(* Logix 5000 project; controller Laser_Cutter vendor 1 type 14 code 149 rev 28.11; software revision 28.00; part 2 of 4 *)
(* tags used below, declared in another part *)
   aBlowOffOnSol : BOOL;
   aBlowoffTimer : TIMER;
   aBoltDriverDownSol : BOOL;
   aBoltDriverUpSol : BOOL;
   aCameraTrigger : BOOL;
   aDoorSafetySwitchUnlockSol : BOOL;
   aExhaustStart : BOOL;
   alarmActive : BOOL;
   automaticSeqStep : DINT;
   autoMode : BOOL;
   autoModeReady : BOOL;
   aWalkingBeamDownSol : BOOL;
   blowoffSeqStep : DINT;
   boltDriverDownDB : TIMER;
   boltDriverSeqStep : DINT;
   boltDriverToStartPOS : BOOL;
   boltDriverToStartPOSdb : TIMER;
   boltDriverUpDB : TIMER;
   Counter : DINT;
   Counter2 : DINT;
   Counter3 : DINT;
   CYCLE_IN_PROG : BOOL;
   cycleTimer : TIMER;
   exeBlowoffSR : BOOL;
   Exec_Bolt_Driver_SR : BOOL;
   Exec_Drive_Bolt : BOOL;
   Exec_Laser_SR : BOOL;
   execLoadPalletSR : BOOL;
   Execute_BlowoffSR : BOOL;
   Execute_MoveToZoneSR : BOOL;
   Execute_VisionInspectionSR : BOOL;
   executeInitializationSequence : BOOL;
   INIT_START_PB : BOOL;
   initDelayTimer : TIMER;
   inspectionSeqStep : DINT;
   LaserSeqStep : INT;
   loadPalletSeqStep : INT;
   MoveToZoneSeqStep : INT;
   p2pCycleTime : TIMER;
   p2pCycleTimeBuffer : DINT;
   readyToMovePallet : BOOL;
   readyToStartCycle : BOOL;
   rejectPartSR : DINT[1];
   runsCompleted : DINT;
   runTime : TIMER;
   startCycleTimer : BOOL;
   startP2PTimer : BOOL;
   startRunTimer : BOOL;
   stationNumber : CONTROL;
   systemInInitializedPosition : BOOL;
   cameraBadPart : ALIAS FOR Local:1:I.Data.8;
   cameraGoodPart : ALIAS FOR Local:1:I.Data.7;
   collarAtStation3 : ALIAS FOR MURR_IMPACT_IO_1:I.Data[1].0;
   collarAtStation4 : ALIAS FOR MURR_IMPACT_IO_1:I.Data[1].1;
   cycleStartPB : ALIAS FOR Local:1:I.Data.3;
   doorOpenedSafetyRelayStatus : ALIAS FOR Local:1:I.Data.1;
   eStopSafetyRelayStatus : ALIAS FOR Local:1:I.Data.0;
   stopPB : ALIAS FOR Local:1:I.Data.4;
(* MainProgram, continued *)

ROUTINE Auto_Seq   (* ladder *)
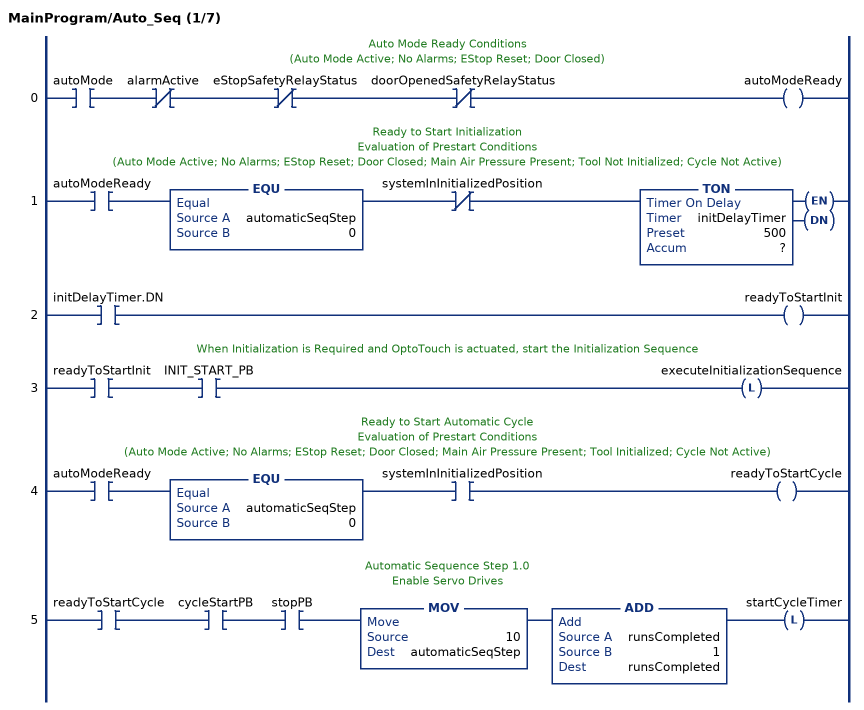
   // Auto Mode Ready Conditions
   // (Auto Mode Active; No Alarms; EStop Reset; Door Closed)
   0: XIC(autoMode)XIO(alarmActive)XIO(eStopSafetyRelayStatus)XIO(doorOpenedSafetyRelayStatus)OTE(autoModeReady);
   // Ready to Start Initialization
   // Evaluation of Prestart Conditions
   // (Auto Mode Active; No Alarms; EStop Reset; Door Closed; Main Air Pressure Present; Tool Not Initialized; Cycle Not Active)
   1: XIC(autoModeReady)EQU(automaticSeqStep,0)XIO(systemInInitializedPosition)TON(initDelayTimer,?,?);
   2: XIC(initDelayTimer.DN)OTE(readyToStartInit);
   // When Initialization is Required and OptoTouch is actuated, start the Initialization Sequence
   3: XIC(readyToStartInit)XIC(INIT_START_PB)OTL(executeInitializationSequence);
   // Ready to Start Automatic Cycle
   // Evaluation of Prestart Conditions
   // (Auto Mode Active; No Alarms; EStop Reset; Door Closed; Main Air Pressure Present; Tool Initialized; Cycle Not Active)
   4: XIC(autoModeReady)EQU(automaticSeqStep,0)XIC(systemInInitializedPosition)OTE(readyToStartCycle);
   // Automatic Sequence Step 1.0
   // Enable Servo Drives
   5: XIC(readyToStartCycle)XIC(cycleStartPB)XIC(stopPB)MOV(10,automaticSeqStep)ADD(runsCompleted,1,runsCompleted)OTL(startCycleTimer);
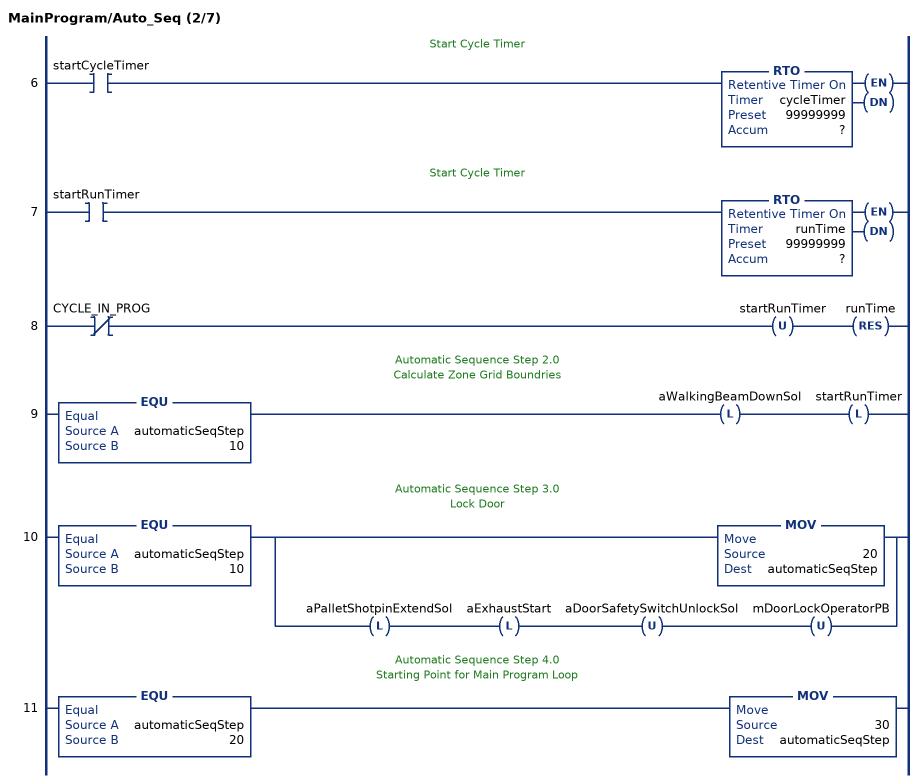
   // Start Cycle Timer
   6: XIC(startCycleTimer)RTO(cycleTimer,?,?);
   // Start Cycle Timer
   7: XIC(startRunTimer)RTO(runTime,?,?);
   8: XIO(CYCLE_IN_PROG)OTU(startRunTimer)RES(runTime);
   // Automatic Sequence Step 2.0
   // Calculate Zone Grid Boundries
   9: EQU(automaticSeqStep,10)OTL(aWalkingBeamDownSol)OTL(startRunTimer);
   // Automatic Sequence Step 3.0
   // Lock Door
   10: EQU(automaticSeqStep,10)[MOV(20,automaticSeqStep) ,OTL(aPalletShotpinExtendSol) OTL(aExhaustStart) OTU(aDoorSafetySwitchUnlockSol) OTU(mDoorLockOperatorPB) ];
   // Automatic Sequence Step 4.0
   // Starting Point for Main Program Loop
   11: EQU(automaticSeqStep,20)MOV(30,automaticSeqStep);
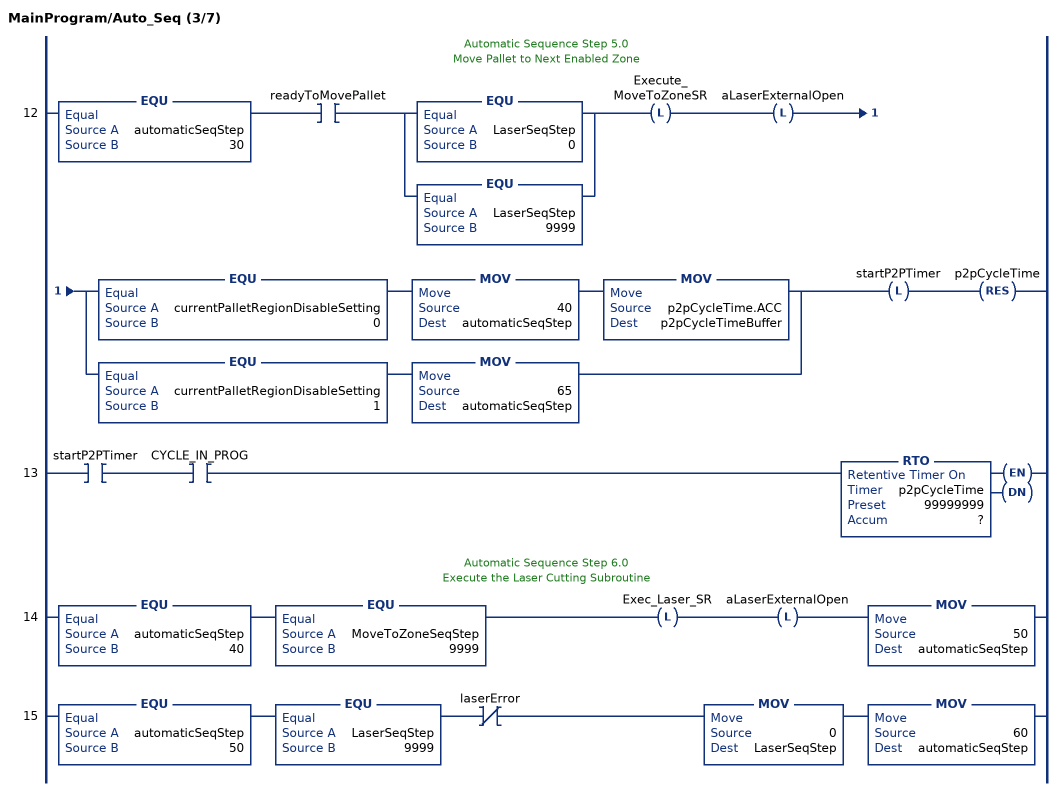
   // Automatic Sequence Step 5.0
   // Move Pallet to Next Enabled Zone
   12: EQU(automaticSeqStep,30)XIC(readyToMovePallet)[EQU(LaserSeqStep,0) ,EQU(LaserSeqStep,9999) ]OTL(Execute_MoveToZoneSR)OTL(aLaserExternalOpen)[EQU(currentPalletRegionDisableSetting,0) MOV(40,automaticSeqStep) MOV(p2pCycleTime.ACC,p2pCycleTimeBuffer) ,EQU(currentPalletRegionDisableSetting,1) MOV(65,automaticSeqStep) ]OTL(startP2PTimer)RES(p2pCycleTime);
   13: XIC(startP2PTimer)XIC(CYCLE_IN_PROG)RTO(p2pCycleTime,?,?);
   // Automatic Sequence Step 6.0
   // Execute the Laser Cutting Subroutine
   14: EQU(automaticSeqStep,40)EQU(MoveToZoneSeqStep,9999)OTL(Exec_Laser_SR)OTL(aLaserExternalOpen)MOV(50,automaticSeqStep);
   15: EQU(automaticSeqStep,50)EQU(LaserSeqStep,9999)XIO(laserError)MOV(0,LaserSeqStep)MOV(60,automaticSeqStep);
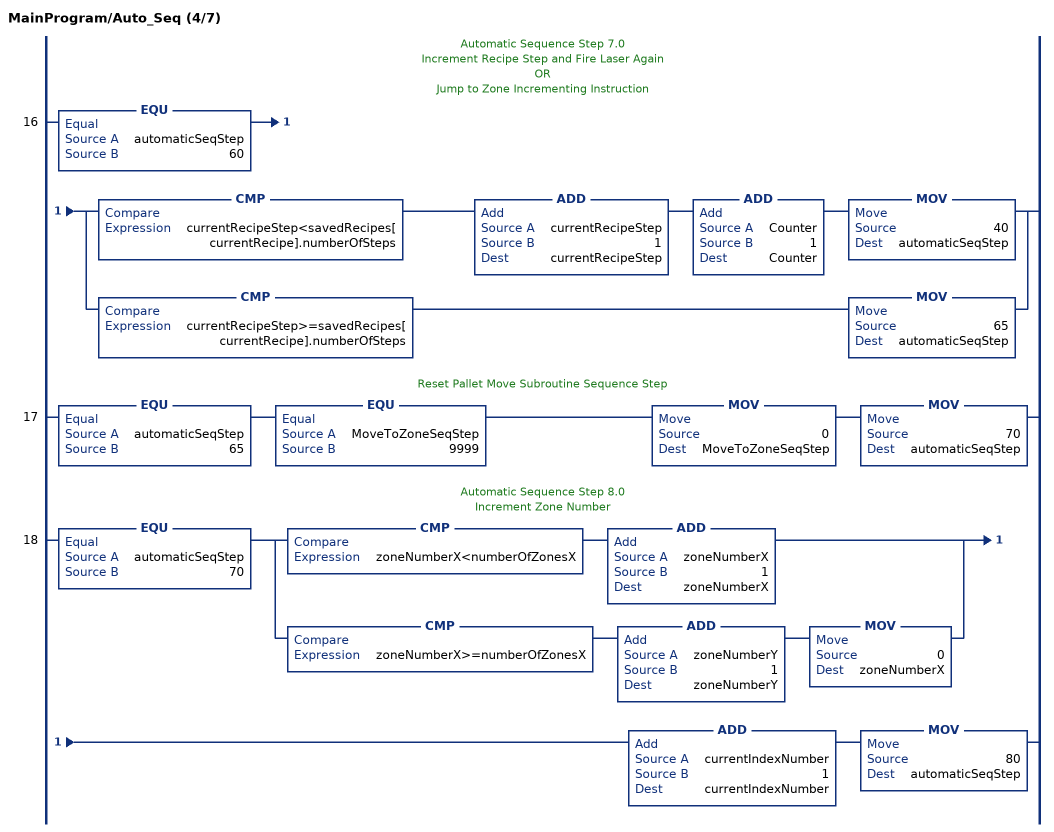
   // Automatic Sequence Step 7.0
   // Increment Recipe Step and Fire Laser Again
   // OR
   // Jump to Zone Incrementing Instruction
   16: EQU(automaticSeqStep,60)[CMP(currentRecipeStep<savedRecipes[currentRecipe].numberOfSteps) ADD(currentRecipeStep,1,currentRecipeStep) ADD(Counter,1,Counter) MOV(40,automaticSeqStep) ,CMP(currentRecipeStep>=savedRecipes[currentRecipe].numberOfSteps) MOV(65,automaticSeqStep) ];
   // Reset Pallet Move Subroutine Sequence Step
   17: EQU(automaticSeqStep,65)EQU(MoveToZoneSeqStep,9999)MOV(0,MoveToZoneSeqStep)MOV(70,automaticSeqStep);
   // Automatic Sequence Step 8.0
   // Increment Zone Number
   18: EQU(automaticSeqStep,70)[CMP(zoneNumberX<numberOfZonesX) ADD(zoneNumberX,1,zoneNumberX) ,CMP(zoneNumberX>=numberOfZonesX) ADD(zoneNumberY,1,zoneNumberY) MOV(0,zoneNumberX) ]ADD(currentIndexNumber,1,currentIndexNumber)MOV(80,automaticSeqStep);
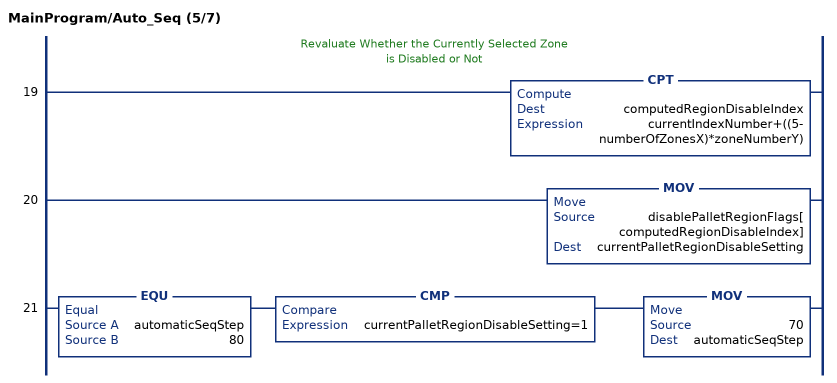
   // Revaluate Whether the Currently Selected Zone
   // is Disabled or Not
   19: CPT(computedRegionDisableIndex,currentIndexNumber+((5-numberOfZonesX)*zoneNumberY));
   20: MOV(disablePalletRegionFlags[computedRegionDisableIndex],currentPalletRegionDisableSetting);
   21: EQU(automaticSeqStep,80)CMP(currentPalletRegionDisableSetting=1)MOV(70,automaticSeqStep);
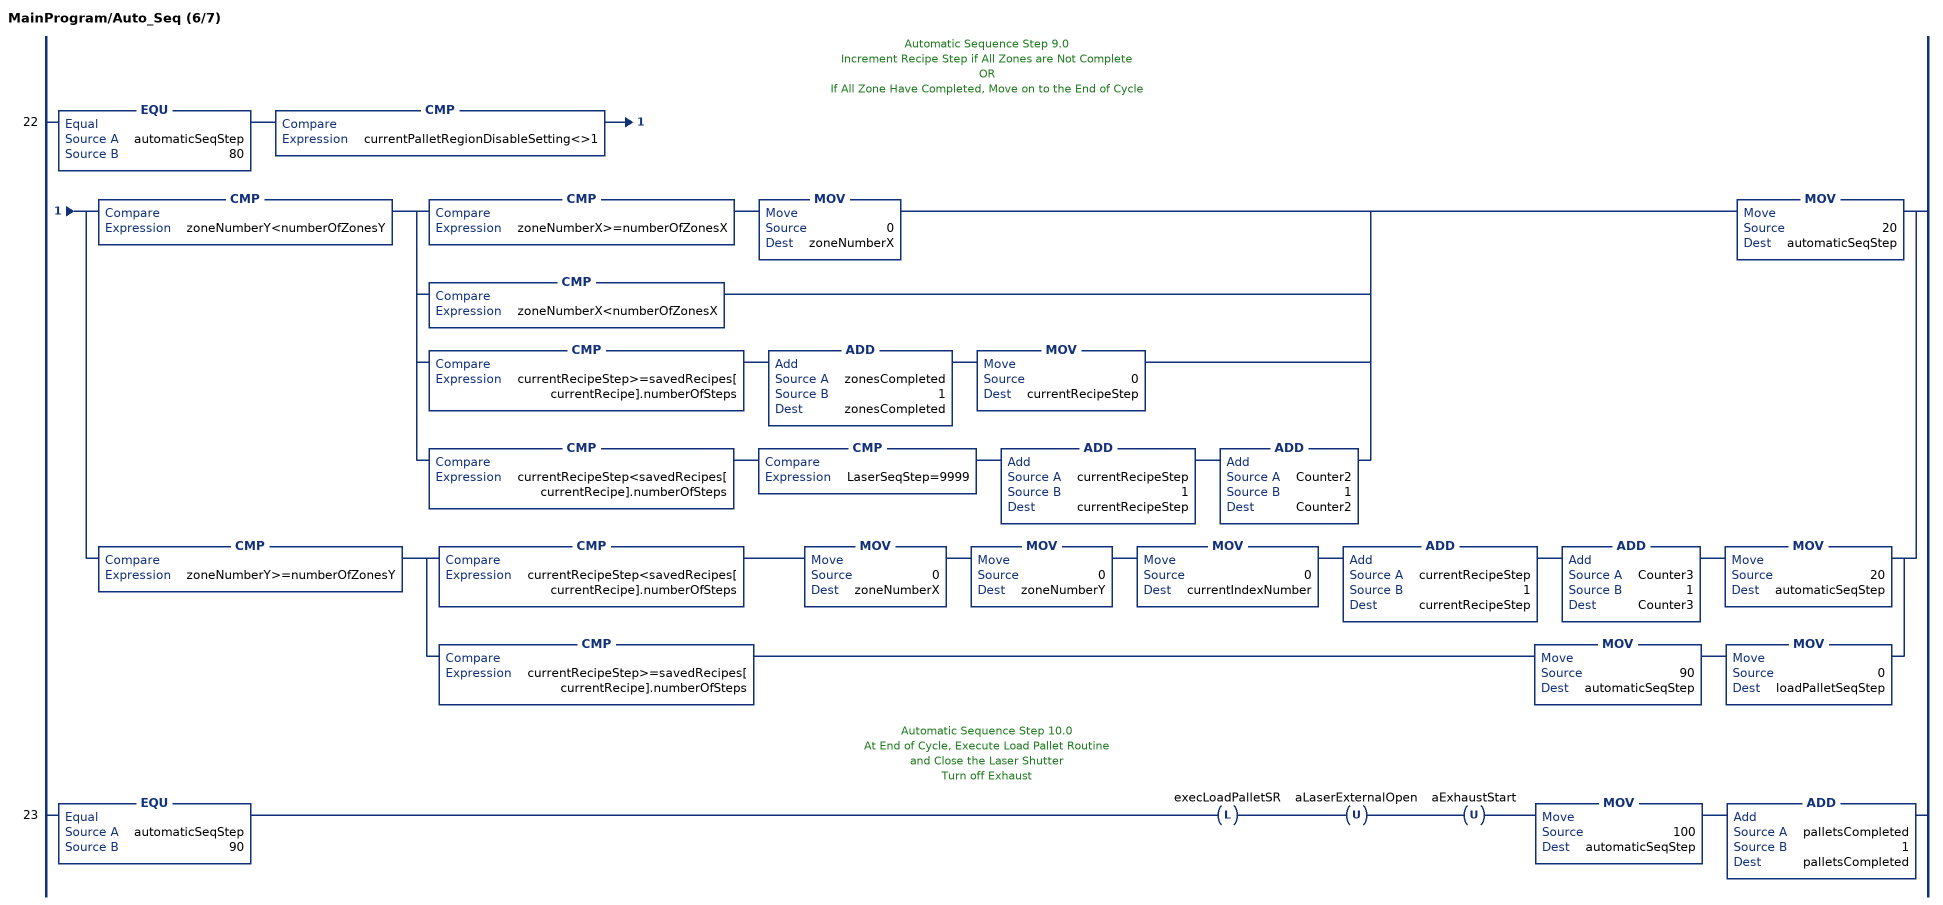
   // Automatic Sequence Step 9.0
   // Increment Recipe Step if All Zones are Not Complete
   // OR
   // If All Zone Have Completed, Move on to the End of Cycle
   22: EQU(automaticSeqStep,80)CMP(currentPalletRegionDisableSetting<>1)[CMP(zoneNumberY<numberOfZonesY) [CMP(zoneNumberX>=numberOfZonesX) MOV(0,zoneNumberX) ,CMP(zoneNumberX<numberOfZonesX) ,[CMP(currentRecipeStep>=savedRecipes[currentRecipe].numberOfSteps) ADD(zonesCompleted,1,zonesCompleted) MOV(0,currentRecipeStep) ,CMP(currentRecipeStep<savedRecipes[currentRecipe].numberOfSteps) CMP(LaserSeqStep=9999) ADD(currentRecipeStep,1,currentRecipeStep) ADD(Counter2,1,Counter2) ] ] MOV(20,automaticSeqStep) ,CMP(zoneNumberY>=numberOfZonesY) [CMP(currentRecipeStep<savedRecipes[currentRecipe].numberOfSteps) MOV(0,zoneNumberX) MOV(0,zoneNumberY) MOV(0,currentIndexNumber) ADD(currentRecipeStep,1,currentRecipeStep) ADD(Counter3,1,Counter3) MOV(20,automaticSeqStep) ,CMP(currentRecipeStep>=savedRecipes[currentRecipe].numberOfSteps) MOV(90,automaticSeqStep) MOV(0,loadPalletSeqStep) ] ];
   // Automatic Sequence Step 10.0
   // At End of Cycle, Execute Load Pallet Routine
   // and Close the Laser Shutter
   // Turn off Exhaust
   23: EQU(automaticSeqStep,90)OTL(execLoadPalletSR)OTU(aLaserExternalOpen)OTU(aExhaustStart)MOV(100,automaticSeqStep)ADD(palletsCompleted,1,palletsCompleted);
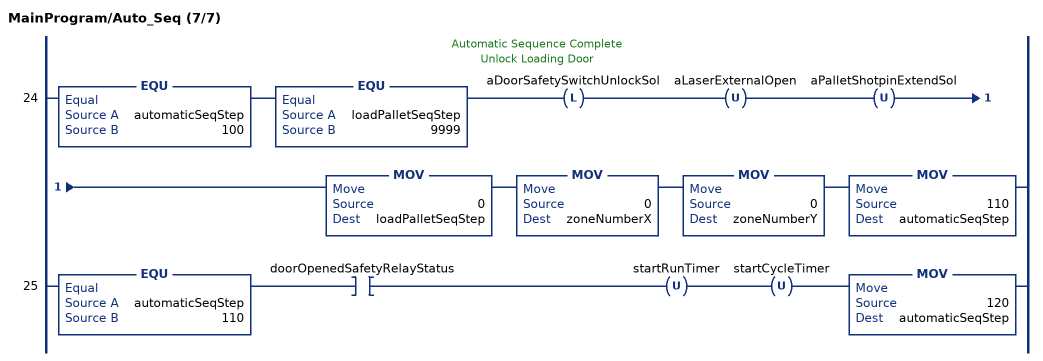
   // Automatic Sequence Complete
   // Unlock Loading Door
   24: EQU(automaticSeqStep,100)EQU(loadPalletSeqStep,9999)OTL(aDoorSafetySwitchUnlockSol)OTU(aLaserExternalOpen)OTU(aPalletShotpinExtendSol)MOV(0,loadPalletSeqStep)MOV(0,zoneNumberX)MOV(0,zoneNumberY)MOV(110,automaticSeqStep);
   25: EQU(automaticSeqStep,110)XIC(doorOpenedSafetyRelayStatus)OTU(startRunTimer)OTU(startCycleTimer)MOV(120,automaticSeqStep);
END_ROUTINE

ROUTINE CycleStations   (* ladder *)
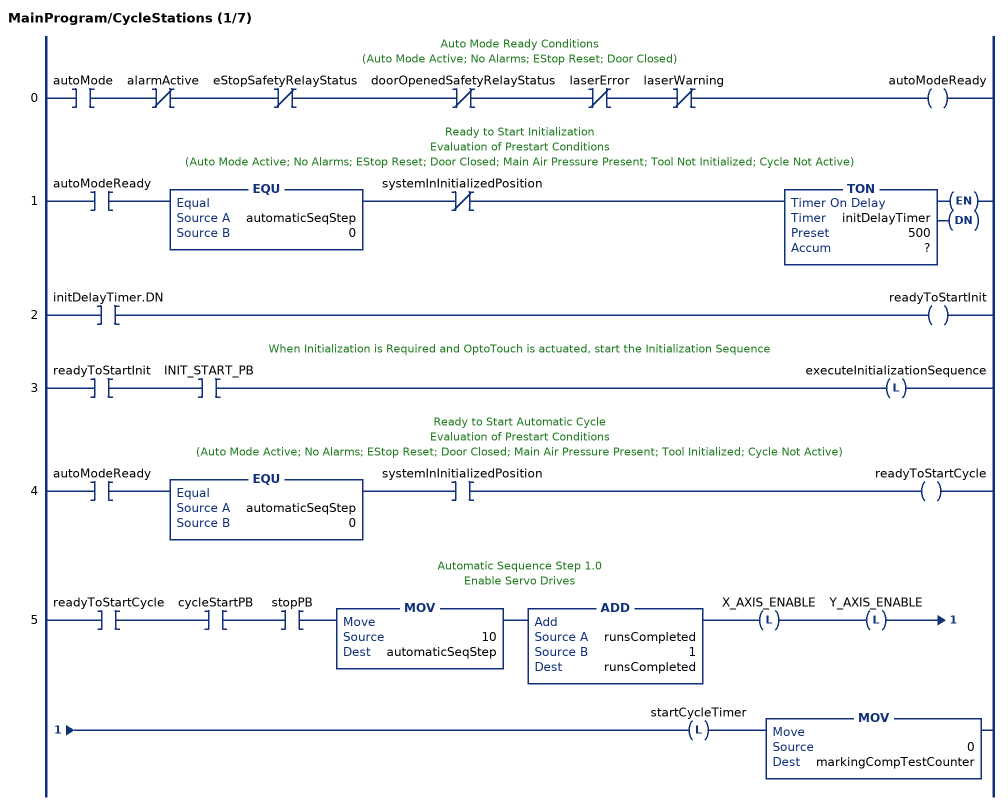
   // Auto Mode Ready Conditions
   // (Auto Mode Active; No Alarms; EStop Reset; Door Closed)
   0: XIC(autoMode)XIO(alarmActive)XIO(eStopSafetyRelayStatus)XIO(doorOpenedSafetyRelayStatus)XIO(laserError)XIO(laserWarning)OTE(autoModeReady);
   // Ready to Start Initialization
   // Evaluation of Prestart Conditions
   // (Auto Mode Active; No Alarms; EStop Reset; Door Closed; Main Air Pressure Present; Tool Not Initialized; Cycle Not Active)
   1: XIC(autoModeReady)EQU(automaticSeqStep,0)XIO(systemInInitializedPosition)TON(initDelayTimer,?,?);
   2: XIC(initDelayTimer.DN)OTE(readyToStartInit);
   // When Initialization is Required and OptoTouch is actuated, start the Initialization Sequence
   3: XIC(readyToStartInit)XIC(INIT_START_PB)OTL(executeInitializationSequence);
   // Ready to Start Automatic Cycle
   // Evaluation of Prestart Conditions
   // (Auto Mode Active; No Alarms; EStop Reset; Door Closed; Main Air Pressure Present; Tool Initialized; Cycle Not Active)
   4: XIC(autoModeReady)EQU(automaticSeqStep,0)XIC(systemInInitializedPosition)OTE(readyToStartCycle);
   // Automatic Sequence Step 1.0
   // Enable Servo Drives
   5: XIC(readyToStartCycle)XIC(cycleStartPB)XIC(stopPB)MOV(10,automaticSeqStep)ADD(runsCompleted,1,runsCompleted)OTL(X_AXIS_ENABLE)OTL(Y_AXIS_ENABLE)OTL(startCycleTimer)MOV(0,markingCompTestCounter);
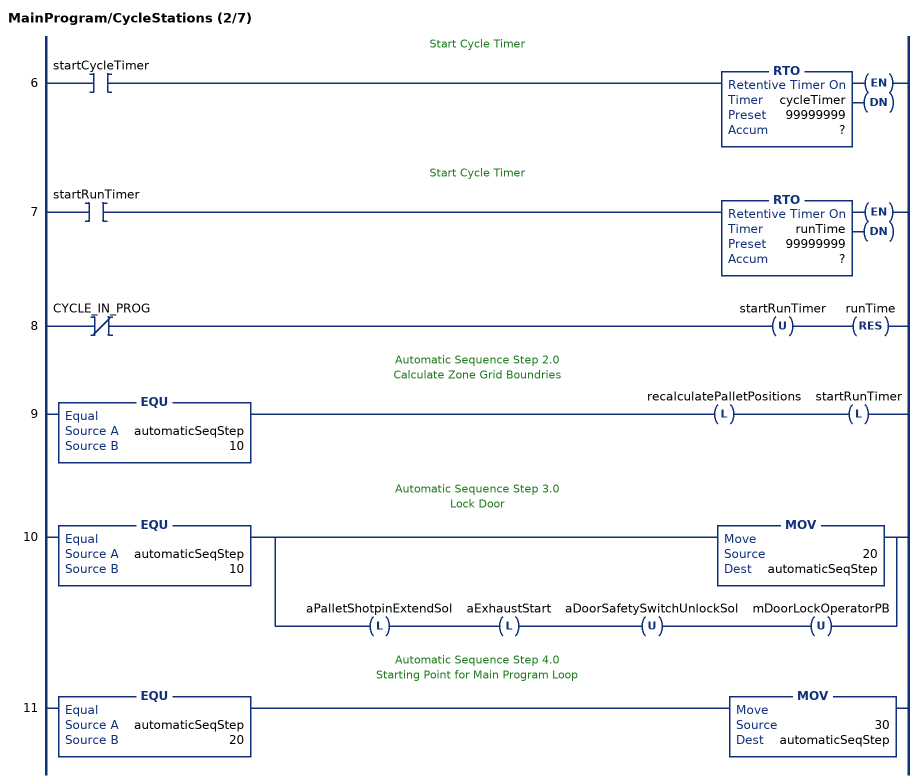
   // Start Cycle Timer
   6: XIC(startCycleTimer)RTO(cycleTimer,?,?);
   // Start Cycle Timer
   7: XIC(startRunTimer)RTO(runTime,?,?);
   8: XIO(CYCLE_IN_PROG)OTU(startRunTimer)RES(runTime);
   // Automatic Sequence Step 2.0
   // Calculate Zone Grid Boundries
   9: EQU(automaticSeqStep,10)OTL(recalculatePalletPositions)OTL(startRunTimer);
   // Automatic Sequence Step 3.0
   // Lock Door
   10: EQU(automaticSeqStep,10)[MOV(20,automaticSeqStep) ,OTL(aPalletShotpinExtendSol) OTL(aExhaustStart) OTU(aDoorSafetySwitchUnlockSol) OTU(mDoorLockOperatorPB) ];
   // Automatic Sequence Step 4.0
   // Starting Point for Main Program Loop
   11: EQU(automaticSeqStep,20)MOV(30,automaticSeqStep);
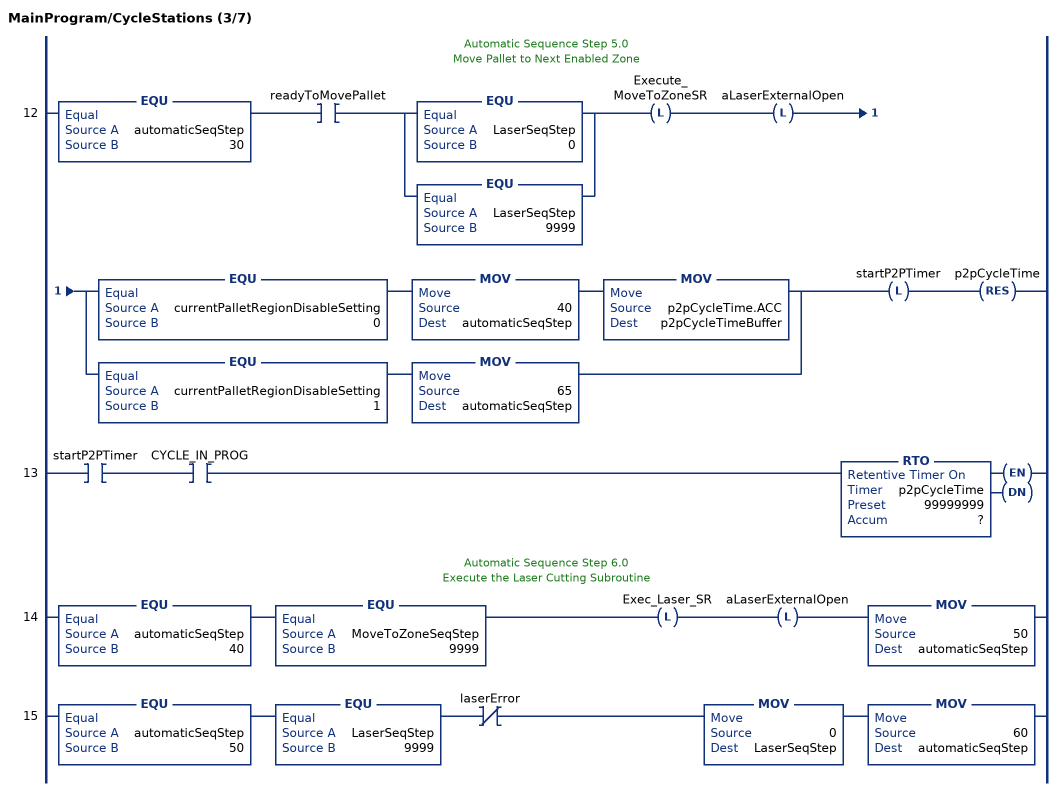
   // Automatic Sequence Step 5.0
   // Move Pallet to Next Enabled Zone
   12: EQU(automaticSeqStep,30)XIC(readyToMovePallet)[EQU(LaserSeqStep,0) ,EQU(LaserSeqStep,9999) ]OTL(Execute_MoveToZoneSR)OTL(aLaserExternalOpen)[EQU(currentPalletRegionDisableSetting,0) MOV(40,automaticSeqStep) MOV(p2pCycleTime.ACC,p2pCycleTimeBuffer) ,EQU(currentPalletRegionDisableSetting,1) MOV(65,automaticSeqStep) ]OTL(startP2PTimer)RES(p2pCycleTime);
   13: XIC(startP2PTimer)XIC(CYCLE_IN_PROG)RTO(p2pCycleTime,?,?);
   // Automatic Sequence Step 6.0
   // Execute the Laser Cutting Subroutine
   14: EQU(automaticSeqStep,40)EQU(MoveToZoneSeqStep,9999)OTL(Exec_Laser_SR)OTL(aLaserExternalOpen)MOV(50,automaticSeqStep);
   15: EQU(automaticSeqStep,50)EQU(LaserSeqStep,9999)XIO(laserError)MOV(0,LaserSeqStep)MOV(60,automaticSeqStep);
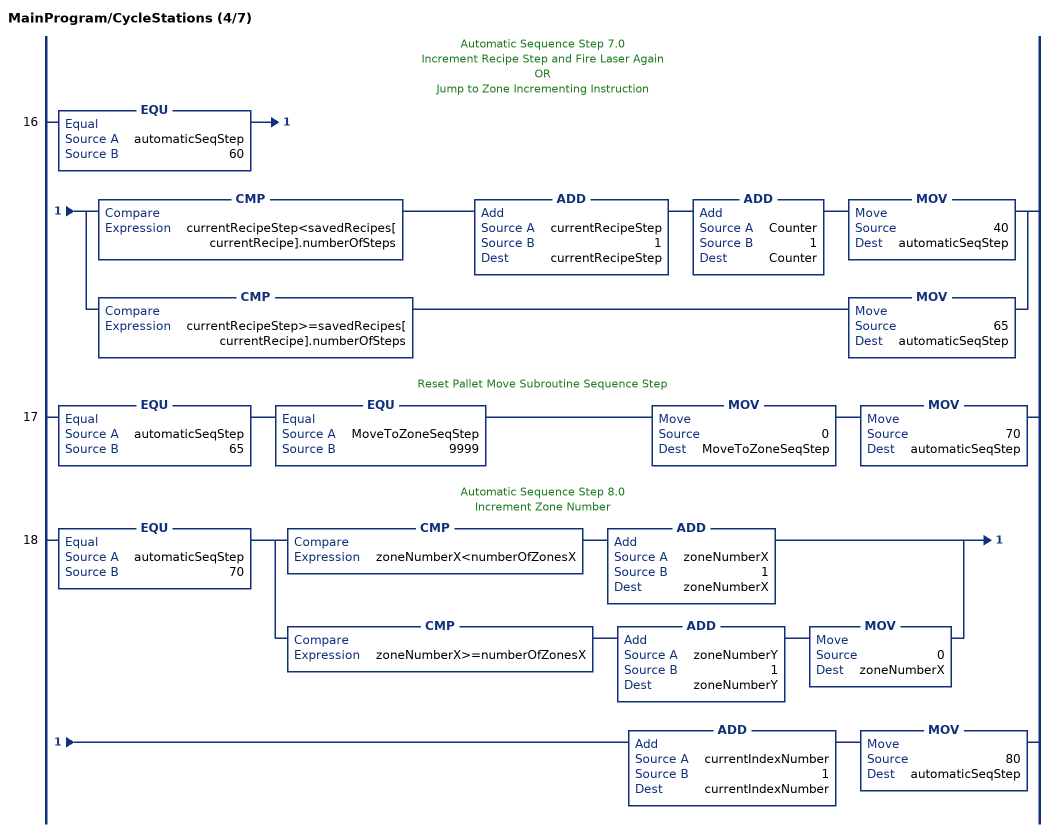
   // Automatic Sequence Step 7.0
   // Increment Recipe Step and Fire Laser Again
   // OR
   // Jump to Zone Incrementing Instruction
   16: EQU(automaticSeqStep,60)[CMP(currentRecipeStep<savedRecipes[currentRecipe].numberOfSteps) ADD(currentRecipeStep,1,currentRecipeStep) ADD(Counter,1,Counter) MOV(40,automaticSeqStep) ,CMP(currentRecipeStep>=savedRecipes[currentRecipe].numberOfSteps) MOV(65,automaticSeqStep) ];
   // Reset Pallet Move Subroutine Sequence Step
   17: EQU(automaticSeqStep,65)EQU(MoveToZoneSeqStep,9999)MOV(0,MoveToZoneSeqStep)MOV(70,automaticSeqStep);
   // Automatic Sequence Step 8.0
   // Increment Zone Number
   18: EQU(automaticSeqStep,70)[CMP(zoneNumberX<numberOfZonesX) ADD(zoneNumberX,1,zoneNumberX) ,CMP(zoneNumberX>=numberOfZonesX) ADD(zoneNumberY,1,zoneNumberY) MOV(0,zoneNumberX) ]ADD(currentIndexNumber,1,currentIndexNumber)MOV(80,automaticSeqStep);
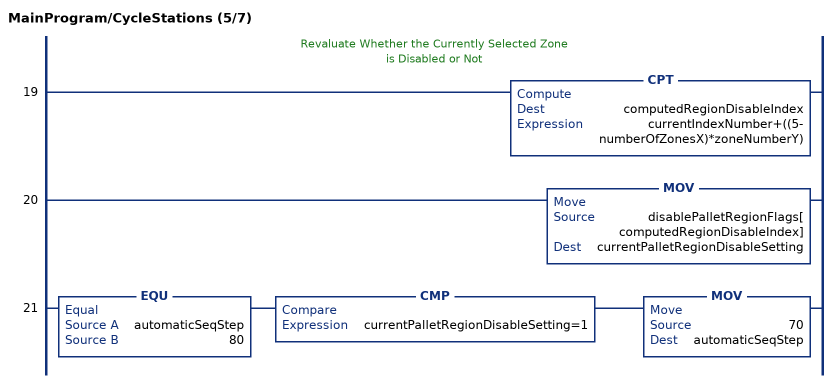
   // Revaluate Whether the Currently Selected Zone
   // is Disabled or Not
   19: CPT(computedRegionDisableIndex,currentIndexNumber+((5-numberOfZonesX)*zoneNumberY));
   20: MOV(disablePalletRegionFlags[computedRegionDisableIndex],currentPalletRegionDisableSetting);
   21: EQU(automaticSeqStep,80)CMP(currentPalletRegionDisableSetting=1)MOV(70,automaticSeqStep);
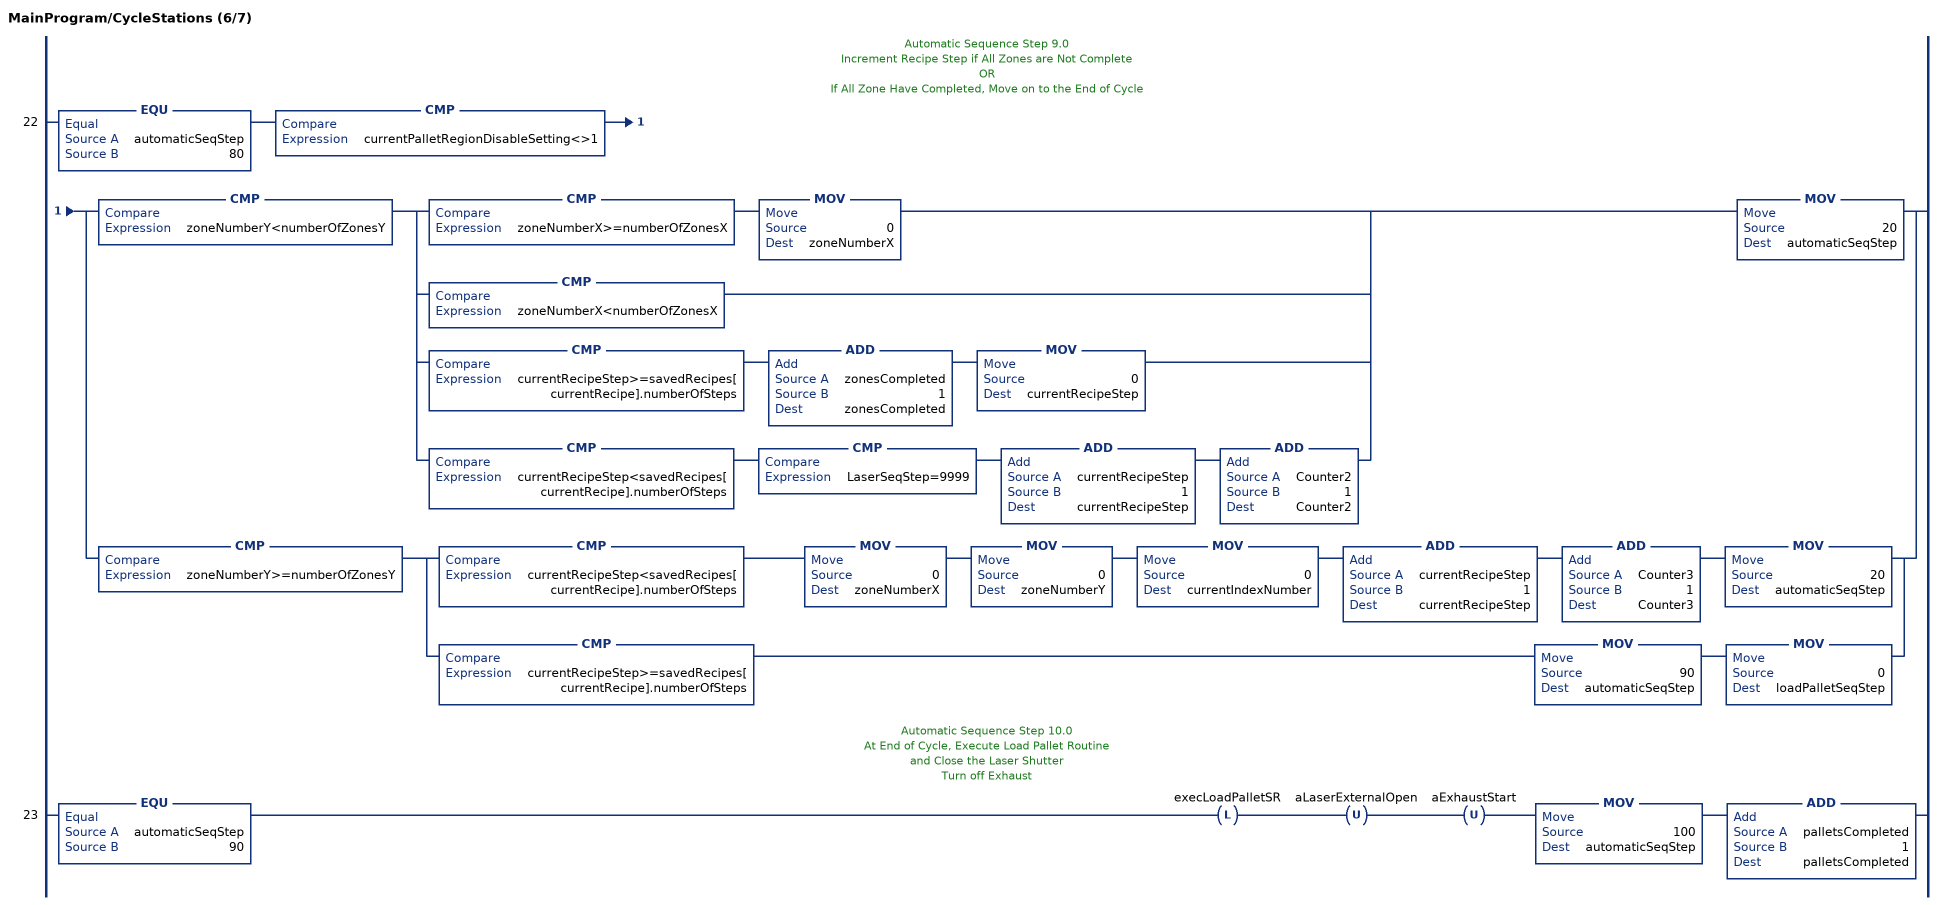
   // Automatic Sequence Step 9.0
   // Increment Recipe Step if All Zones are Not Complete
   // OR
   // If All Zone Have Completed, Move on to the End of Cycle
   22: EQU(automaticSeqStep,80)CMP(currentPalletRegionDisableSetting<>1)[CMP(zoneNumberY<numberOfZonesY) [CMP(zoneNumberX>=numberOfZonesX) MOV(0,zoneNumberX) ,CMP(zoneNumberX<numberOfZonesX) ,[CMP(currentRecipeStep>=savedRecipes[currentRecipe].numberOfSteps) ADD(zonesCompleted,1,zonesCompleted) MOV(0,currentRecipeStep) ,CMP(currentRecipeStep<savedRecipes[currentRecipe].numberOfSteps) CMP(LaserSeqStep=9999) ADD(currentRecipeStep,1,currentRecipeStep) ADD(Counter2,1,Counter2) ] ] MOV(20,automaticSeqStep) ,CMP(zoneNumberY>=numberOfZonesY) [CMP(currentRecipeStep<savedRecipes[currentRecipe].numberOfSteps) MOV(0,zoneNumberX) MOV(0,zoneNumberY) MOV(0,currentIndexNumber) ADD(currentRecipeStep,1,currentRecipeStep) ADD(Counter3,1,Counter3) MOV(20,automaticSeqStep) ,CMP(currentRecipeStep>=savedRecipes[currentRecipe].numberOfSteps) MOV(90,automaticSeqStep) MOV(0,loadPalletSeqStep) ] ];
   // Automatic Sequence Step 10.0
   // At End of Cycle, Execute Load Pallet Routine
   // and Close the Laser Shutter
   // Turn off Exhaust
   23: EQU(automaticSeqStep,90)OTL(execLoadPalletSR)OTU(aLaserExternalOpen)OTU(aExhaustStart)MOV(100,automaticSeqStep)ADD(palletsCompleted,1,palletsCompleted);
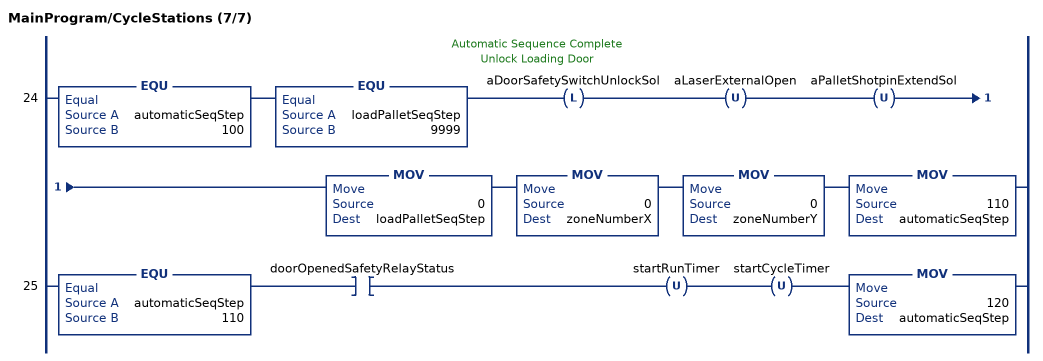
   // Automatic Sequence Complete
   // Unlock Loading Door
   24: EQU(automaticSeqStep,100)EQU(loadPalletSeqStep,9999)OTL(aDoorSafetySwitchUnlockSol)OTU(aLaserExternalOpen)OTU(aPalletShotpinExtendSol)MOV(0,loadPalletSeqStep)MOV(0,zoneNumberX)MOV(0,zoneNumberY)MOV(110,automaticSeqStep);
   25: EQU(automaticSeqStep,110)XIC(doorOpenedSafetyRelayStatus)OTU(startRunTimer)OTU(startCycleTimer)MOV(120,automaticSeqStep);
END_ROUTINE

ROUTINE Exec_Blowoff_SR   (* ladder *)
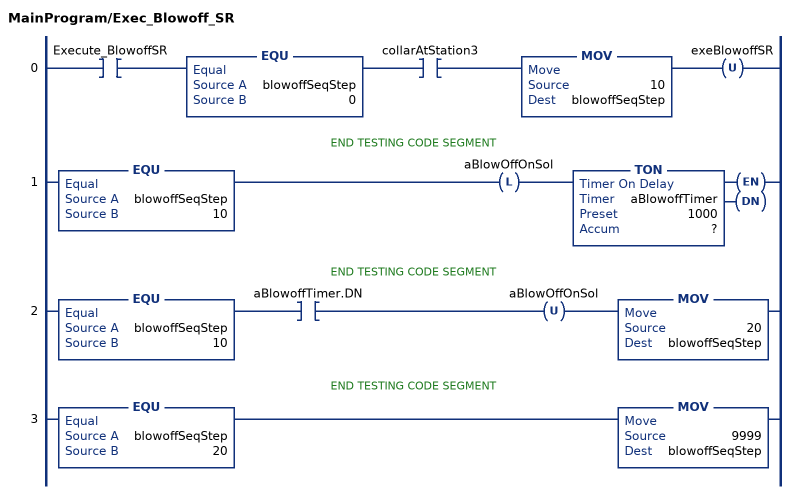
   0: XIC(Execute_BlowoffSR)EQU(blowoffSeqStep,0)XIC(collarAtStation3)MOV(10,blowoffSeqStep)OTU(exeBlowoffSR);
   // END TESTING CODE SEGMENT
   1: EQU(blowoffSeqStep,10)OTL(aBlowOffOnSol)TON(aBlowoffTimer,?,?);
   // END TESTING CODE SEGMENT
   2: EQU(blowoffSeqStep,10)XIC(aBlowoffTimer.DN)OTU(aBlowOffOnSol)MOV(20,blowoffSeqStep);
   // END TESTING CODE SEGMENT
   3: EQU(blowoffSeqStep,20)MOV(9999,blowoffSeqStep);
END_ROUTINE

ROUTINE Exec_Bolt_Driver_SR   (* ladder *)
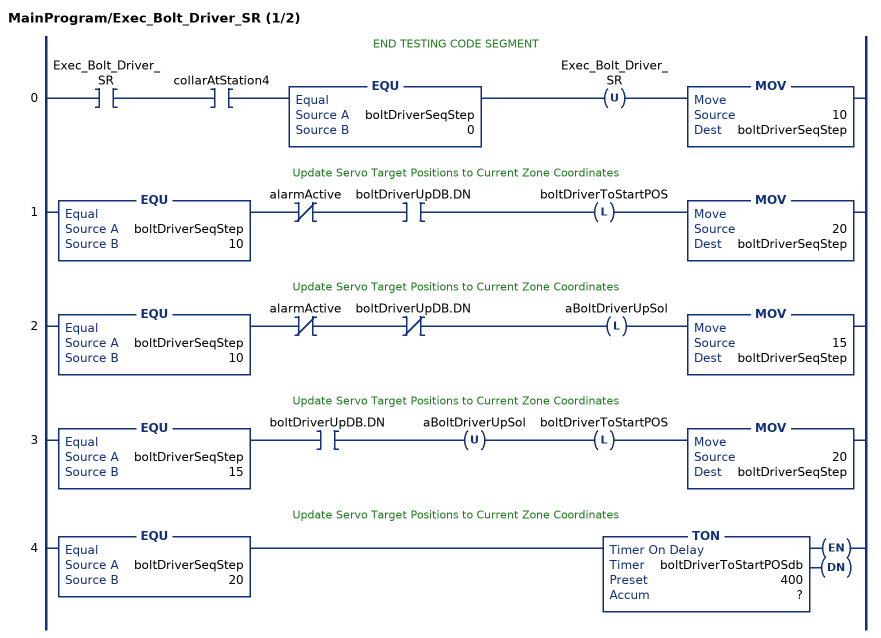
   // END TESTING CODE SEGMENT
   0: XIC(Exec_Bolt_Driver_SR)XIC(collarAtStation4)EQU(boltDriverSeqStep,0)OTU(Exec_Bolt_Driver_SR)MOV(10,boltDriverSeqStep);
   // Update Servo Target Positions to Current Zone Coordinates
   1: EQU(boltDriverSeqStep,10)XIO(alarmActive)XIC(boltDriverUpDB.DN)OTL(boltDriverToStartPOS)MOV(20,boltDriverSeqStep);
   // Update Servo Target Positions to Current Zone Coordinates
   2: EQU(boltDriverSeqStep,10)XIO(alarmActive)XIO(boltDriverUpDB.DN)OTL(aBoltDriverUpSol)MOV(15,boltDriverSeqStep);
   // Update Servo Target Positions to Current Zone Coordinates
   3: EQU(boltDriverSeqStep,15)XIC(boltDriverUpDB.DN)OTU(aBoltDriverUpSol)OTL(boltDriverToStartPOS)MOV(20,boltDriverSeqStep);
   // Update Servo Target Positions to Current Zone Coordinates
   4: EQU(boltDriverSeqStep,20)TON(boltDriverToStartPOSdb,?,?);
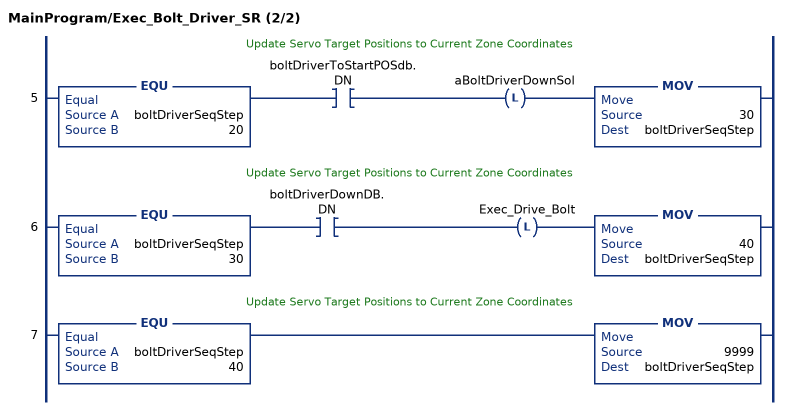
   // Update Servo Target Positions to Current Zone Coordinates
   5: EQU(boltDriverSeqStep,20)XIC(boltDriverToStartPOSdb.DN)OTL(aBoltDriverDownSol)MOV(30,boltDriverSeqStep);
   // Update Servo Target Positions to Current Zone Coordinates
   6: EQU(boltDriverSeqStep,30)XIC(boltDriverDownDB.DN)OTL(Exec_Drive_Bolt)MOV(40,boltDriverSeqStep);
   // Update Servo Target Positions to Current Zone Coordinates
   7: EQU(boltDriverSeqStep,40)MOV(9999,boltDriverSeqStep);
END_ROUTINE

ROUTINE Exec_Inspection_SR   (* ladder *)
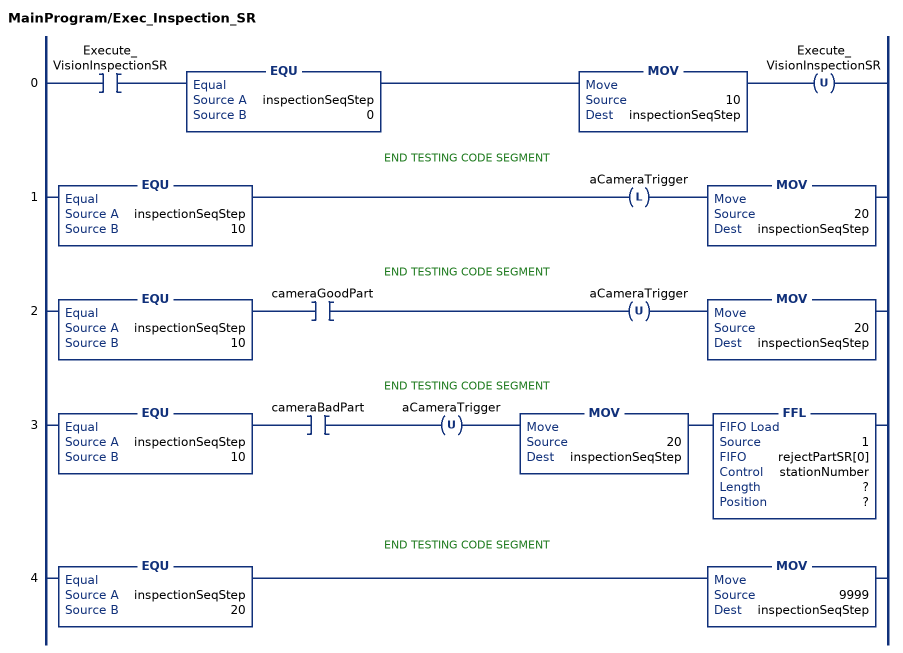
   0: XIC(Execute_VisionInspectionSR)EQU(inspectionSeqStep,0)MOV(10,inspectionSeqStep)OTU(Execute_VisionInspectionSR);
   // END TESTING CODE SEGMENT
   1: EQU(inspectionSeqStep,10)OTL(aCameraTrigger)MOV(20,inspectionSeqStep);
   // END TESTING CODE SEGMENT
   2: EQU(inspectionSeqStep,10)XIC(cameraGoodPart)OTU(aCameraTrigger)MOV(20,inspectionSeqStep);
   // END TESTING CODE SEGMENT
   3: EQU(inspectionSeqStep,10)XIC(cameraBadPart)OTU(aCameraTrigger)MOV(20,inspectionSeqStep)FFL(1,rejectPartSR[0],stationNumber,?,?);
   // END TESTING CODE SEGMENT
   4: EQU(inspectionSeqStep,20)MOV(9999,inspectionSeqStep);
END_ROUTINE
